{attribute 'qualified_only'}
{attribute 'strict'}
TYPE E_InterlockType :
(
	RunInterlock,
	StartPermissive,
	StopPermissive
);
END_TYPE

(* stored: Version 1.1.0.1, ProductVersion 3.1.4024.12
   DUT E_InterlockType: Id {8fed1186-f6a6-434d-905f-4c89e3f7a7d1} *)
